//{attribute 'qualified_only'}
VAR_GLOBAL
	robot1, robot2 : RobotA21;
	toolStorageA21Left, toolStorageA21Right : A21ToolStorage;
	
	skidA21Left, skidA21Right : SkidMagazine;
	
	stagingTableLeft, stagingTableRight : WoodBunkTable;
	magazineA21Left, magazineA21Right : SkidMagazine;
	
	strapperA21 : StrapMachine;
	
	horizontalDriveA21Left, horizontalDriveA21Right : AirPiston;
	verticalDriveA21Left, verticalDriveA21Right : ClearLinkMC;
	pistonA21Bottom : SimplePiston;
	
	suctionA21Top : ARRAY[1..3] OF SuctionPad;
	suctionA21Left : ARRAY[1..4] OF SuctionPad;
	suctionA21Right : ARRAY[1..4] OF SuctionPad; 
	suctionA21Bottom : ARRAY[1..2] OF SuctionPad;
END_VAR

(* stored: Version 1.1.0.1, ProductVersion 3.1.4024.11
   GVL Hardware: Id {72ad6a3a-e035-4ae1-b9b7-c68bdd948b2f} *)
